FUNCTION_BLOCK FB_Conveyor
VAR_INPUT
	stInput	:ST_ConveyorInputs;
END_VAR
VAR_OUTPUT
	stOutput	:ST_ConveyorOutputs;
END_VAR
VAR
	eActConveyorState	:E_ConveyorState	:= E_ConveyorState.INIT;
	bPartDetected		:BOOL	:=FALSE;
END_VAR

A_ProcessFlow();

ACTION A_ProcessFlow:
CASE eActConveyorState OF 
	E_ConveyorState.INIT:
		// When conveyor part is at the end of the conveyor stop it. robot will clear the part
		IF M_PartDetectedAtEnd() THEN
			eActConveyorState := E_ConveyorState.STOP;
		END_IF
		
		// When part is not at the end, start the conveyor to move 
		IF NOT M_PartDetectedAtEnd()  AND NOT stInput.bRobInSpace THEN
			IF P_GetPart2Move THEN
				eActConveyorState	:= E_ConveyorState.REQUEST_MOVE;
			END_IF
		END_IF
	
		
		
	E_ConveyorState.REQUEST_MOVE:
		stOutput.bMoveConveyor := TRUE;
		eActConveyorState	:= E_ConveyorState.MOVING;
		
		
		
	E_ConveyorState.MOVING:
		IF P_GetConveyorMoving THEN
			// DO Nothing. Wait here until Part is detected
			
		END_IF
		IF M_PartDetectedAtEnd() THEN
			eActConveyorState	:= E_ConveyorState.STOP;
		END_IF
		
		
		
	E_ConveyorState.STOP:
		stOutput.bMoveConveyor := FALSE;
		IF NOT P_GetConveyorMoving THEN
			// DO Nothing
			eActConveyorState	:= E_ConveyorState.INIT;
		ELSE
			eActConveyorState	:= E_ConveyorState.ERROR;
		END_IF
		
		
		
	E_ConveyorState.ERROR:
		// TODO: Wait for Error Handling
		
END_CASE

bPartDetected	:= M_PartDetectedAtEnd();
END_ACTION

METHOD M_PartDetectedAtEnd : BOOL
VAR_INPUT
END_VAR
M_PartDetectedAtEnd := stInput.bPartDetected;
RETURN;
END_METHOD

PROPERTY P_GetConveyorMoving : BOOL
GET
stInput.bConveyorIsMoving := stOutput.bMoveConveyor;
END_GET
END_PROPERTY

PROPERTY P_GetPart2Move : BOOL
GET
P_GetPart2Move := GVL_IO.Conveyor_Inputs.bPartAvailable2Move;
END_GET
END_PROPERTY

END_FUNCTION_BLOCK

(* stored: Version 1.1.0.1, ProductVersion 3.1.4024.16
   POU FB_Conveyor: Id {d8956dc1-793f-4c9c-be4b-5c7e93e0da86}, SpecialFunc None
   Action A_ProcessFlow: Id {8534e87c-3222-459b-82b1-d9cf51637e16}
   Method M_PartDetectedAtEnd: Id {033389a7-cb82-4909-8ee7-94f6f4b7144c}
   Property P_GetConveyorMoving: Id {38eb1a51-4cc6-4443-87f3-9ada5fc322ca}
   Get Get: Id {88b9459f-a7e3-4b98-bad0-22c92405af84}
   Property P_GetPart2Move: Id {af88d269-f469-4ffb-afc7-9947117517bd}
   Get Get: Id {0bfb4706-9db3-4ce6-81eb-8f2e7bca6fe0} *)
